PROGRAM Tiersheet_Car
VAR
	TiersheetRemoverTMR: TOF;
	TrolleySlowUnlatch: TOF;
	VacTog: TOGGLE;
	SGE: TOGGLE;
	SGR: TOGGLE;

	TrolleyToSheetBin_F: BOOL;
	TrolleyToHoist_FR: BOOL;
	TrolleyToSheetBin_FR: BOOL;
	TrolleyToFrameBin_F: BOOL;
	TrolleytoHoist: BOOL;
	TrolleytoSheetBin: BOOL;
	TrolleytoFrameBin: BOOL;
	TiersheetCarriage_Auto: BOOL;
	sCarriageAuto: BOOL;
	TierCar_Tog: TOGGLE;
	sCurrent_Loc: REAL;
	sRequested_Loc: REAL;
	TrolleytoHoistSlowdown: BOOL;
	On_Loc: BOOL;
	Direction: BOOL;
	Reverse: BOOL;
	Forward: BOOL;
	t1: BOOL;
	t2: BOOL;
	t3: BOOL;
	t4: BOOL;
	t5: BOOL;
	t6: BOOL;
	L6: BOOL;
	L4: BOOL;
	L2: BOOL;
	L1: BOOL;
	Slow: BOOL;
	SlowR: BOOL;
	vactest: BOOL;
	Routine_Move_HoistToBin: BOOL;
	TiersheetRemoverTMR2: TOF;
	HoistToBin_Delay: TON;

	FrameRemover_TOG: TOGGLE;
	FrameRemoverPulse: TP;

	FrameClampsTOG: TOGGLE;
	FrameClampPulse: TP;


	At_TopFrame: BOOL;
	Gripper_Release_Pulse: TP;
	Gripper_Release_Delay: TON;
	ToSheetBinDelay: TON;

	TopFrame_Removal: BOOL;
	FrameLockPulse: TP;
	ToFrameBinDelay: TON;
	ToSheetBinDelay2: TON;




	Frame_PickUp: BOOL;
	Removal_Pulse: TP;
	Release_Delay: TON;


	Carriage_Extended_Latch: BOOL;
	Test: BOOL;
	Trolly_Delay: TON;
	TestTroley: Toggle;
	Delay: TON;
	sbTest: BOOL;
END_VAR
VAR // added by the converter: edge detectors and wires of the graphical bodies
    _w1, _w2, _w3, _w4, _w5, _w6, _w7, _w8, _w9 : INT;
    _w10, _w11 : BOOL;
END_VAR

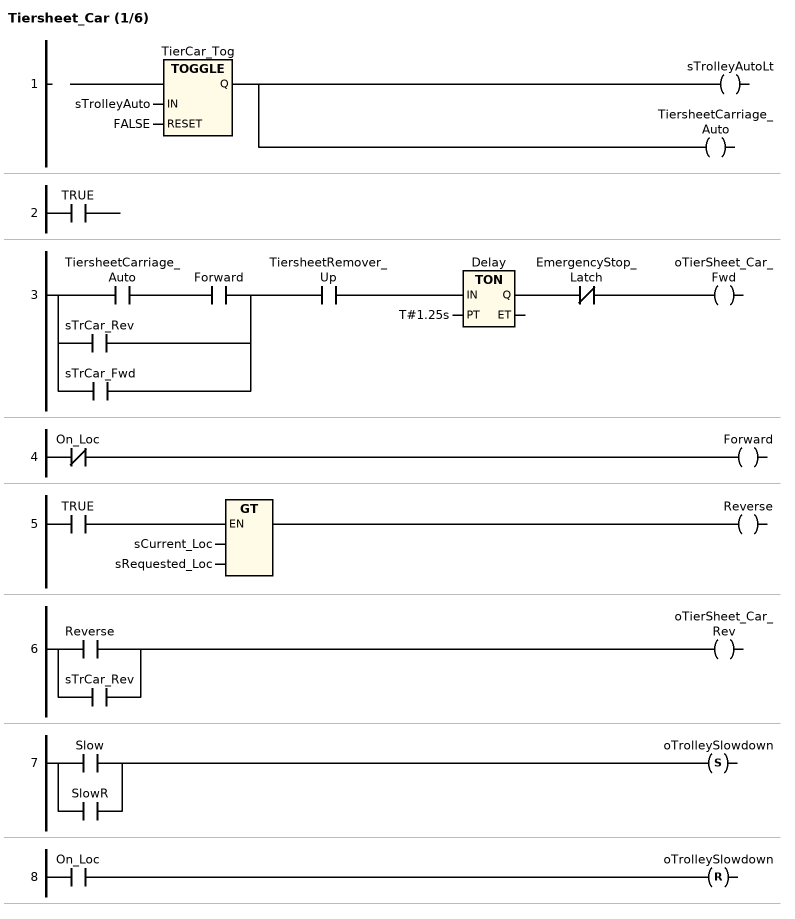
// NETWORK 1
TierCar_Tog(IN := sTrolleyAuto, RESET := FALSE); // TOGGLE
sTrolleyAutoLt := TierCar_Tog.Q;
TiersheetCarriage_Auto := TierCar_Tog.Q;

// NETWORK 2

// NETWORK 3
Delay(IN := (TiersheetCarriage_Auto AND Forward OR sTrCar_Rev OR sTrCar_Fwd) AND TiersheetRemover_Up, PT := T#1.25s); // TON
oTierSheet_Car_Fwd := Delay.Q AND NOT EmergencyStop_Latch;

// NETWORK 4
Forward := NOT On_Loc;

// NETWORK 5
Reverse := sCurrent_Loc > sRequested_Loc;

// NETWORK 6
oTierSheet_Car_Rev := Reverse OR sTrCar_Rev;

// NETWORK 7
oTrolleySlowdown S= Slow OR SlowR;

// NETWORK 8
oTrolleySlowdown R= On_Loc;

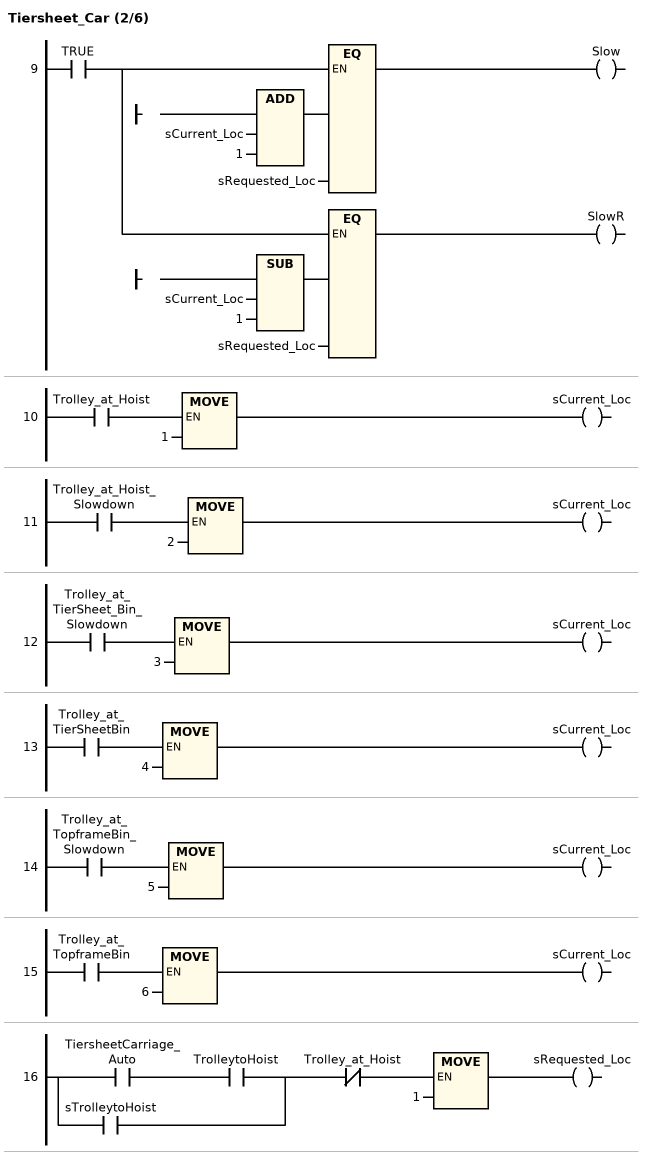
// NETWORK 9
Slow := sCurrent_Loc + 1 = sRequested_Loc;
SlowR := sCurrent_Loc - 1 = sRequested_Loc;

// NETWORK 10
IF Trolley_at_Hoist THEN _w1 := 1; END_IF
sCurrent_Loc := _w1;

// NETWORK 11
IF Trolley_at_Hoist_Slowdown THEN _w2 := 2; END_IF
sCurrent_Loc := _w2;

// NETWORK 12
IF Trolley_at_TierSheet_Bin_Slowdown THEN _w3 := 3; END_IF
sCurrent_Loc := _w3;

// NETWORK 13
IF Trolley_at_TierSheetBin THEN _w4 := 4; END_IF
sCurrent_Loc := _w4;

// NETWORK 14
IF Trolley_at_TopframeBin_Slowdown THEN _w5 := 5; END_IF
sCurrent_Loc := _w5;

// NETWORK 15
IF Trolley_at_TopframeBin THEN _w6 := 6; END_IF
sCurrent_Loc := _w6;

// NETWORK 16
IF (TiersheetCarriage_Auto AND TrolleytoHoist OR sTrolleytoHoist) AND NOT Trolley_at_Hoist THEN _w7 := 1; END_IF
sRequested_Loc := _w7;

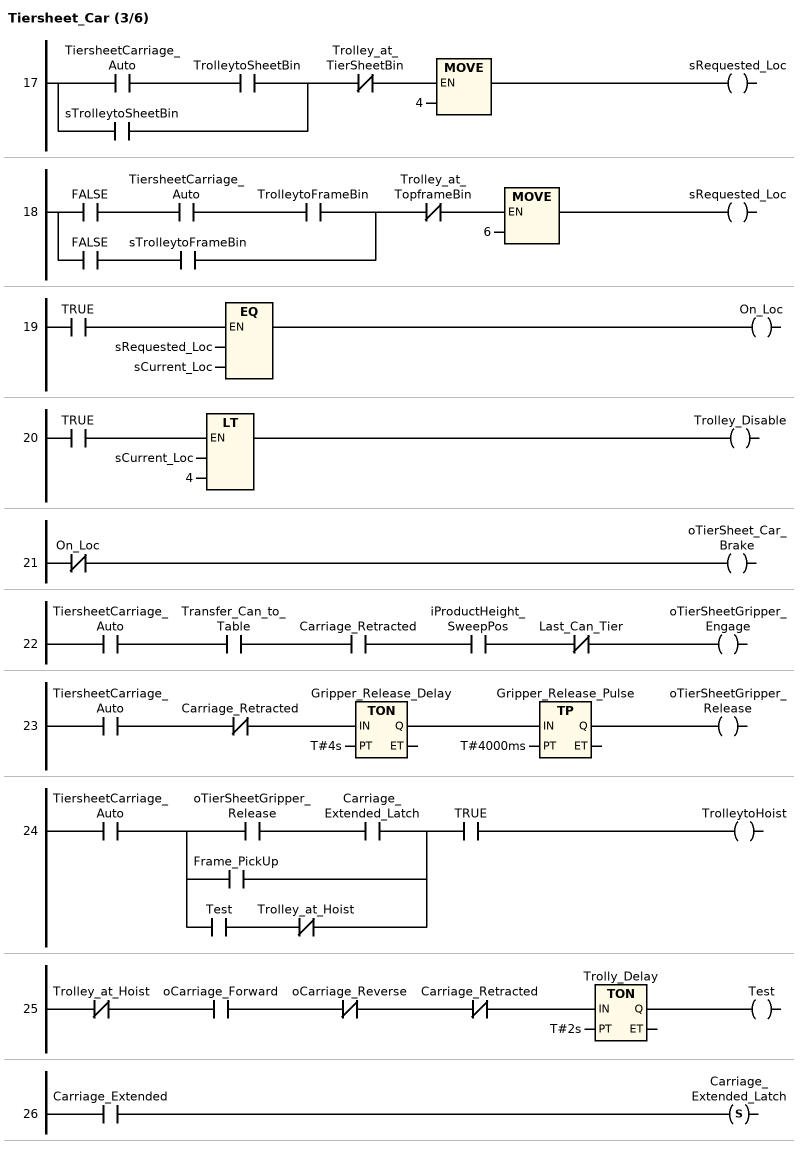
// NETWORK 17
IF (TiersheetCarriage_Auto AND TrolleytoSheetBin OR sTrolleytoSheetBin) AND NOT Trolley_at_TierSheetBin THEN
    _w8 := 4;
END_IF
sRequested_Loc := _w8;

// NETWORK 18
IF (FALSE AND TiersheetCarriage_Auto AND TrolleytoFrameBin OR FALSE AND sTrolleytoFrameBin) AND NOT Trolley_at_TopframeBin THEN
    _w9 := 6;
END_IF
sRequested_Loc := _w9;

// NETWORK 19
On_Loc := sRequested_Loc = sCurrent_Loc;

// NETWORK 20
Trolley_Disable := sCurrent_Loc < 4;

// NETWORK 21
oTierSheet_Car_Brake := NOT On_Loc;

// NETWORK 22
oTierSheetGripper_Engage := TiersheetCarriage_Auto AND Transfer_Can_to_Table AND Carriage_Retracted AND iProductHeight_SweepPos AND NOT Last_Can_Tier;

// NETWORK 23
Gripper_Release_Delay(IN := TiersheetCarriage_Auto AND NOT Carriage_Retracted, PT := T#4s); // TON
Gripper_Release_Pulse(IN := Gripper_Release_Delay.Q, PT := T#4000ms); // TP
oTierSheetGripper_Release := Gripper_Release_Pulse.Q;

// NETWORK 24
TrolleytoHoist := (TiersheetCarriage_Auto AND (oTierSheetGripper_Release AND Carriage_Extended_Latch OR Frame_PickUp OR Test AND NOT Trolley_at_Hoist)) AND TRUE;

// NETWORK 25
Trolly_Delay(IN := NOT Trolley_at_Hoist AND oCarriage_Forward AND NOT oCarriage_Reverse AND NOT Carriage_Retracted, PT := T#2s); // TON
Test := Trolly_Delay.Q;

// NETWORK 26
Carriage_Extended_Latch S= Carriage_Extended;

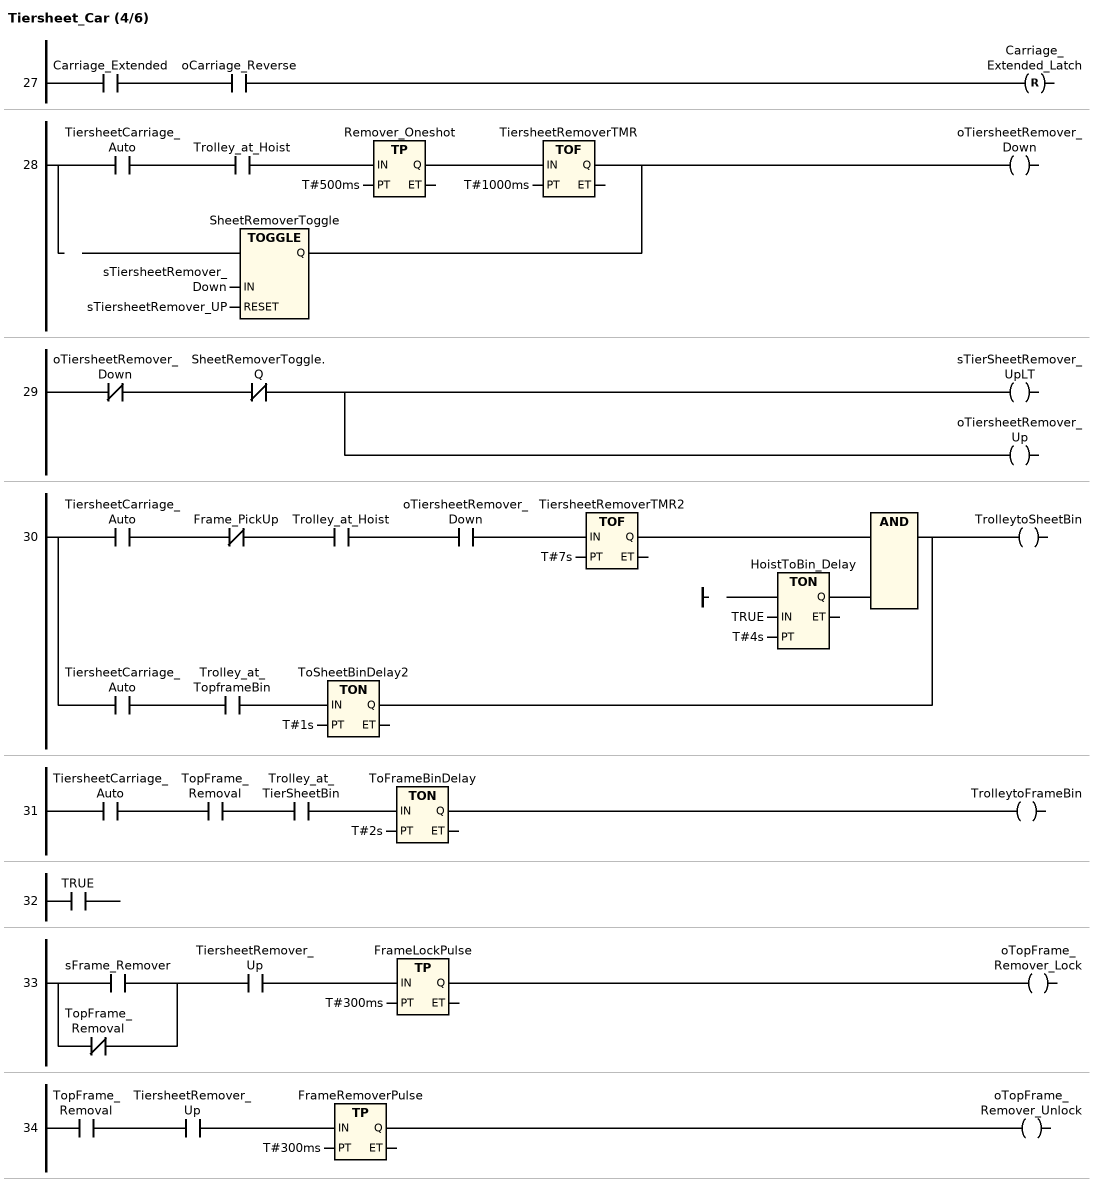
// NETWORK 27
Carriage_Extended_Latch R= Carriage_Extended AND oCarriage_Reverse;

// NETWORK 28
Remover_Oneshot(IN := TiersheetCarriage_Auto AND Trolley_at_Hoist, PT := T#500ms); // TP
TiersheetRemoverTMR(IN := Remover_Oneshot.Q, PT := T#1000ms); // TOF
SheetRemoverToggle(IN := sTiersheetRemover_Down, RESET := sTiersheetRemover_UP); // TOGGLE
oTiersheetRemover_Down := TiersheetRemoverTMR.Q OR SheetRemoverToggle.Q;

// NETWORK 29
_w10 := NOT oTiersheetRemover_Down AND NOT SheetRemoverToggle.Q;
sTierSheetRemover_UpLT := _w10;
oTiersheetRemover_Up := _w10;

// NETWORK 30
TiersheetRemoverTMR2(IN := TiersheetCarriage_Auto AND (NOT Frame_PickUp AND Trolley_at_Hoist AND oTiersheetRemover_Down), PT := T#7s); // TOF
HoistToBin_Delay(IN := TRUE, PT := T#4s); // TON
ToSheetBinDelay2(IN := TiersheetCarriage_Auto AND Trolley_at_TopframeBin, PT := T#1s); // TON
TrolleytoSheetBin := TiersheetRemoverTMR2.Q AND HoistToBin_Delay.Q OR ToSheetBinDelay2.Q;

// NETWORK 31
ToFrameBinDelay(IN := TiersheetCarriage_Auto AND TopFrame_Removal AND Trolley_at_TierSheetBin, PT := T#2s); // TON
TrolleytoFrameBin := ToFrameBinDelay.Q;

// NETWORK 32

// NETWORK 33
FrameLockPulse(IN := (sFrame_Remover OR NOT TopFrame_Removal) AND TiersheetRemover_Up, PT := T#300ms); // TP
oTopFrame_Remover_Lock := FrameLockPulse.Q;

// NETWORK 34
FrameRemoverPulse(IN := TopFrame_Removal AND TiersheetRemover_Up, PT := T#300ms); // TP
oTopFrame_Remover_Unlock := FrameRemoverPulse.Q;

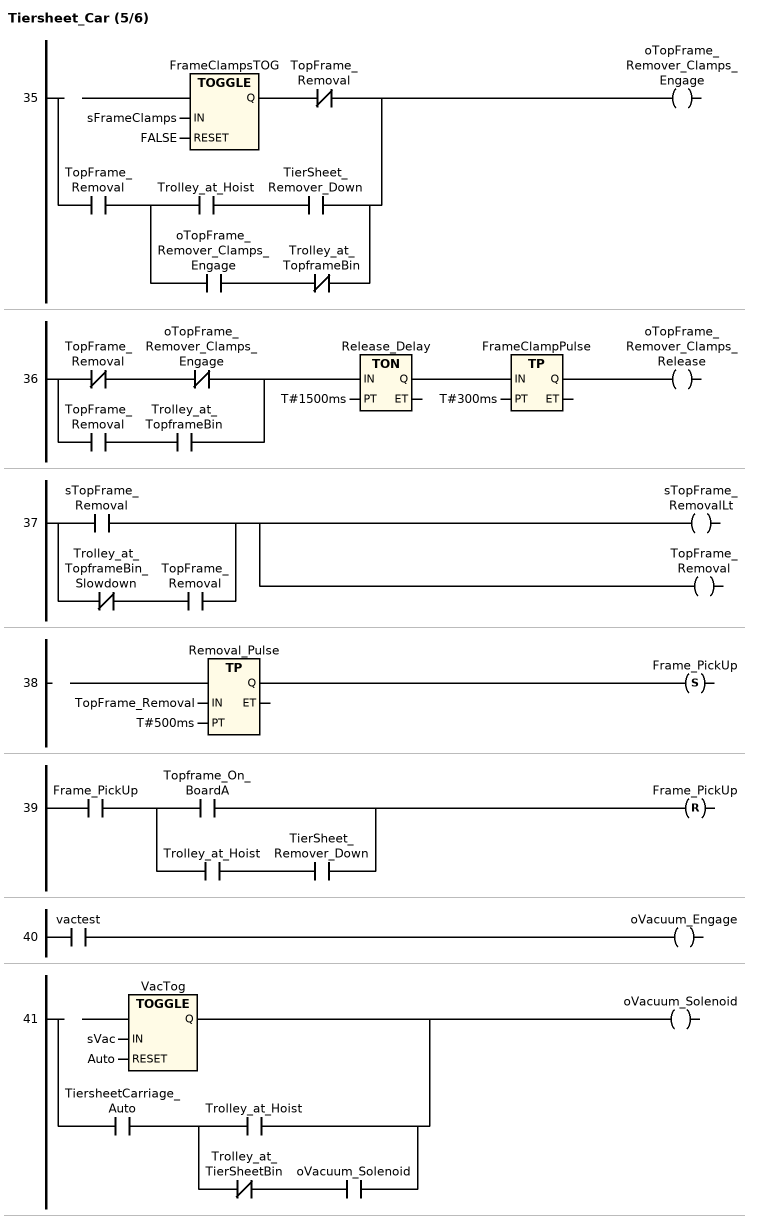
// NETWORK 35
FrameClampsTOG(IN := sFrameClamps, RESET := FALSE); // TOGGLE
oTopFrame_Remover_Clamps_Engage := FrameClampsTOG.Q AND NOT TopFrame_Removal OR TopFrame_Removal AND (Trolley_at_Hoist AND TierSheet_Remover_Down OR oTopFrame_Remover_Clamps_Engage AND NOT Trolley_at_TopframeBin);

// NETWORK 36
Release_Delay(IN := NOT TopFrame_Removal AND NOT oTopFrame_Remover_Clamps_Engage OR TopFrame_Removal AND Trolley_at_TopframeBin, PT := T#1500ms); // TON
FrameClampPulse(IN := Release_Delay.Q, PT := T#300ms); // TP
oTopFrame_Remover_Clamps_Release := FrameClampPulse.Q;

// NETWORK 37
_w11 := sTopFrame_Removal OR NOT Trolley_at_TopframeBin_Slowdown AND TopFrame_Removal;
sTopFrame_RemovalLt := _w11;
TopFrame_Removal := _w11;

// NETWORK 38
Removal_Pulse(IN := TopFrame_Removal, PT := T#500ms); // TP
Frame_PickUp S= Removal_Pulse.Q;

// NETWORK 39
Frame_PickUp R= Frame_PickUp AND (Topframe_On_BoardA OR Trolley_at_Hoist AND TierSheet_Remover_Down);

// NETWORK 40
oVacuum_Engage := vactest;

// NETWORK 41
VacTog(IN := sVac, RESET := Auto); // TOGGLE
oVacuum_Solenoid := VacTog.Q OR TiersheetCarriage_Auto AND (Trolley_at_Hoist OR NOT Trolley_at_TierSheetBin AND oVacuum_Solenoid);

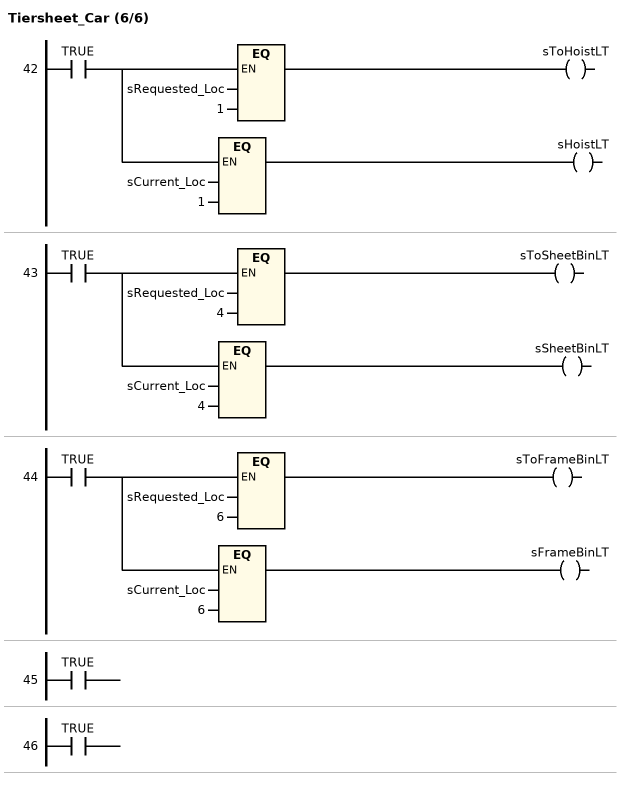
// NETWORK 42
sToHoistLT := sRequested_Loc = 1;
sHoistLT := sCurrent_Loc = 1;

// NETWORK 43
sToSheetBinLT := sRequested_Loc = 4;
sSheetBinLT := sCurrent_Loc = 4;

// NETWORK 44
sToFrameBinLT := sRequested_Loc = 6;
sFrameBinLT := sCurrent_Loc = 6;

// NETWORK 45

// NETWORK 46

END_PROGRAM

(* stored: Version 1.1.0.1, ProductVersion 3.1.4024.16
   POU Tiersheet_Car: Id {4af457df-2145-42e1-ab6f-dc3052639f80}, SpecialFunc None *)
